FUNCTION_BLOCK plant
  (* Standard: 61499-2 *)
  (* Version 0.1, 2017-00-25, hpea485, UOA *)
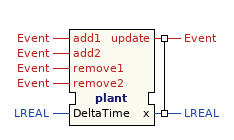
  EVENT_INPUT
    add1;
    add2;
    remove1;
    remove2;
  END_EVENT
  EVENT_OUTPUT
    update WITH x;
  END_EVENT
  VAR_INPUT
    DeltaTime : LREAL := 0.01;
  END_VAR
  VAR_OUTPUT
    x : LREAL;
  END_VAR
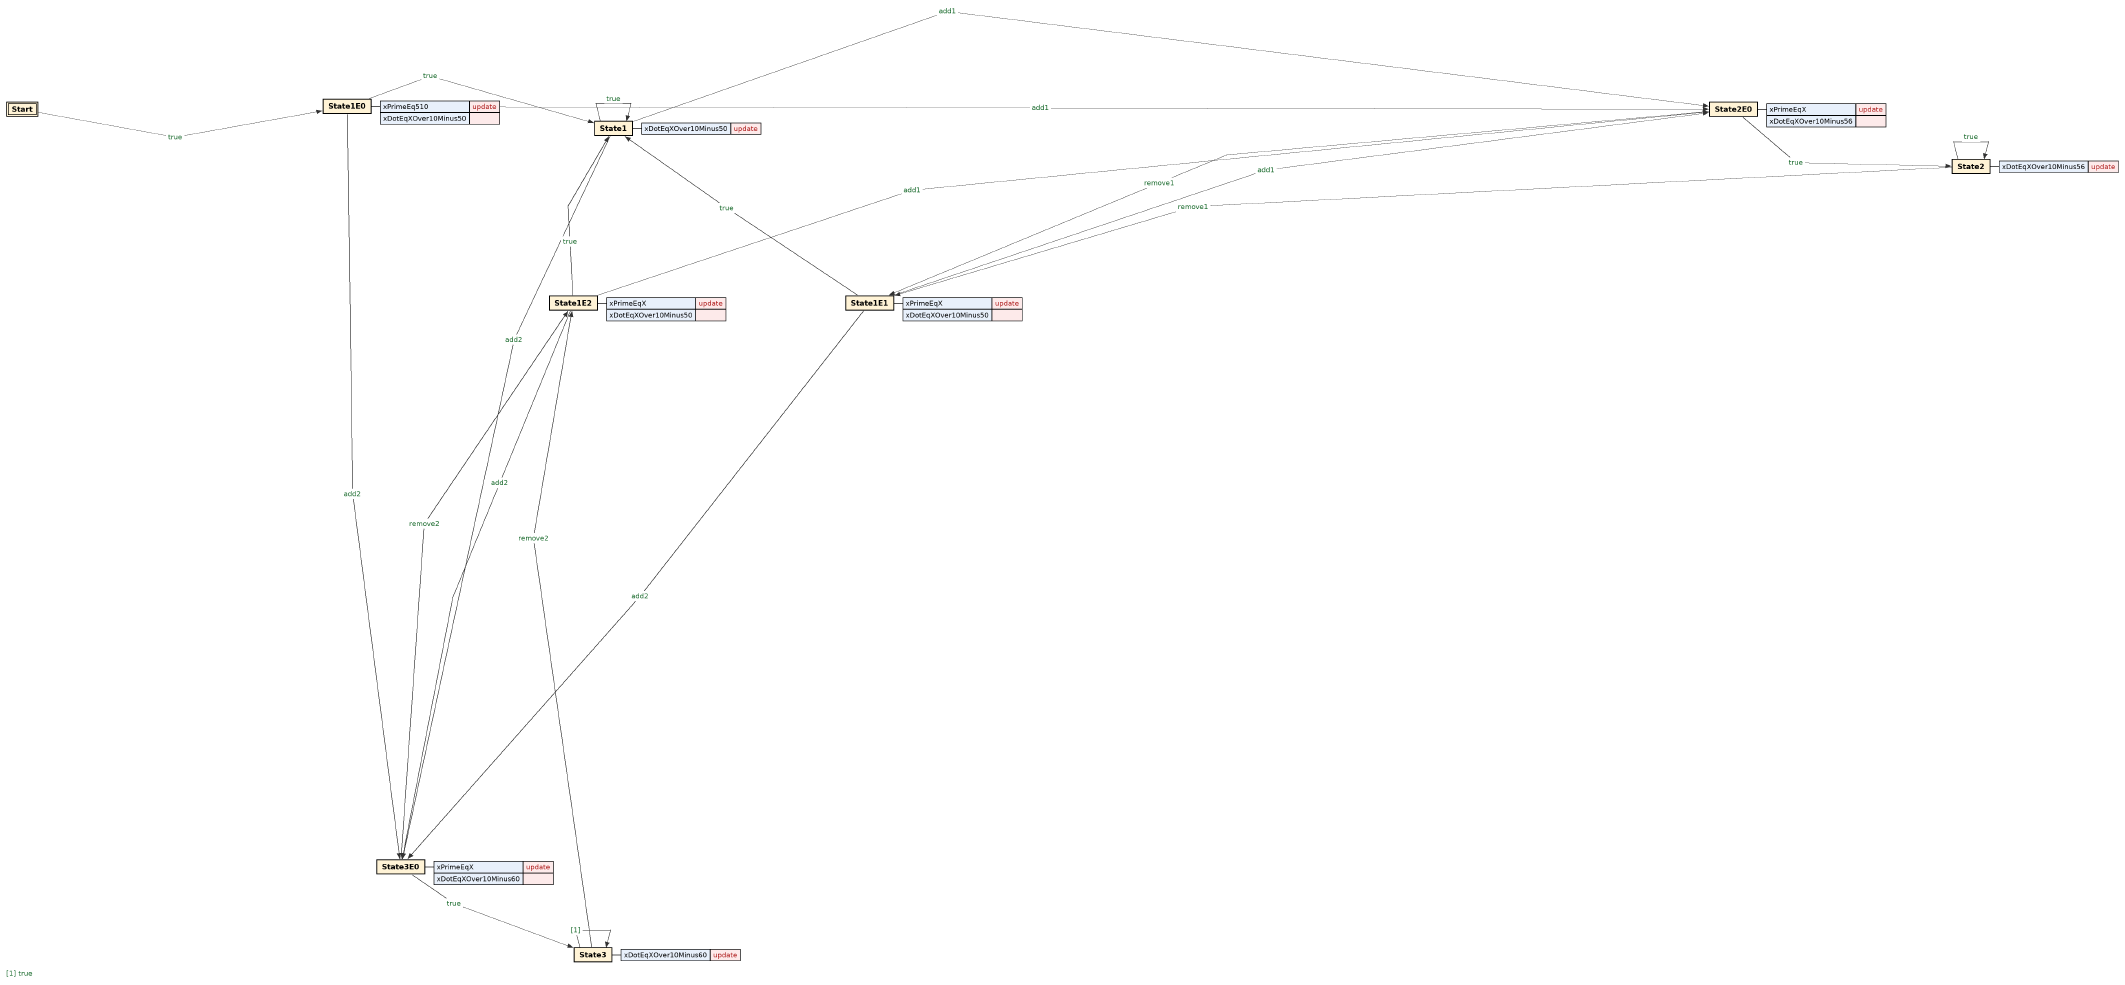
  EC_STATES
    Start;
    State1E0 : xPrimeEq510 -> update, xDotEqXOver10Minus50;
    State1 : xDotEqXOver10Minus50 -> update;
    State2E0 : xPrimeEqX -> update, xDotEqXOver10Minus56;
    State2 : xDotEqXOver10Minus56 -> update;
    State1E1 : xPrimeEqX -> update, xDotEqXOver10Minus50;
    State3E0 : xPrimeEqX -> update, xDotEqXOver10Minus60;
    State3 : xDotEqXOver10Minus60 -> update;
    State1E2 : xPrimeEqX -> update, xDotEqXOver10Minus50;
  END_STATES
  EC_TRANSITIONS
    Start TO State1E0 := true;
    State1E0 TO State2E0 := add1;
    State1E0 TO State3E0 := add2;
    State1E0 TO State1 := true;
    State1 TO State2E0 := add1;
    State1 TO State3E0 := add2;
    State1 TO State1 := true;
    State2E0 TO State1E1 := remove1;
    State2E0 TO State2 := true;
    State2 TO State1E1 := remove1;
    State2 TO State2 := true;
    State1E1 TO State2E0 := add1;
    State1E1 TO State3E0 := add2;
    State1E1 TO State1 := true;
    State3E0 TO State1E2 := remove2;
    State3E0 TO State3 := true;
    State3 TO State1E2 := remove2;
    State3 TO State3 := true;
    State1E2 TO State2E0 := add1;
    State1E2 TO State3E0 := add2;
    State1E2 TO State1 := true;
  END_TRANSITIONS
  ALGORITHM xPrimeEq510 IN C: (* ODE_init *)
x_prime = 510;
  END_ALGORITHM
  ALGORITHM xPrimeEqX IN C: (* ODE_init *)
x_prime = x;
  END_ALGORITHM
  ALGORITHM xDotEqXOver10Minus50 IN C: (* ODE *)
x_dot = (x / 10) - 50;
  END_ALGORITHM
  ALGORITHM xDotEqXOver10Minus56 IN C: (* ODE *)
x_dot = (x / 10) - 56;
  END_ALGORITHM
  ALGORITHM xDotEqXOver10Minus60 IN C: (* ODE *)
x_dot = (x / 10) - 60;
  END_ALGORITHM
END_FUNCTION_BLOCK
